{attribute 'GeneratedUsingTerminal: EJ9576-0000-0019'}
{attribute addProperty BoxType "EJ9576-0000-0019"}
{attribute addProperty Description "EJ9576 Brake chopper terminal"}
{attribute addProperty Physics "KK"}
{attribute addProperty Id "BCT_InputsAT %I*BCT_Inputs_4B98789517WcStateAT %I*WcState_9091E0EB2InfoDataAT %I*InfoData_32EB74EA10"}
{attribute addProperty CRC "2242598916"}
{attribute addProperty Size "29"}
TYPE EJ9576_85AB5804 EXTENDS EtcSlaveTerminalBase_947E5A46 :
STRUCT
	{attribute addProperty Name "BCT_Inputs"}
	BCT_Inputs : BCT_Inputs_4B987895;
	{attribute addProperty Name "WcState"}
	WcState : WcState_9091E0EB;
	{attribute addProperty Name "InfoData"}
	InfoData : InfoData_32EB74EA;
END_STRUCT
END_TYPE

(* stored: Version 1.2.0.0, ProductVersion 3.1.4024.9
   DUT EJ9576_85AB5804: Id {afaedde1-d663-4784-bcf0-ec9d6cfdf188} *)
